{attribute 'qualified_only'}
VAR_GLOBAL
	// PLC Rack
	// Digital Outputs
	bTest					 AT %Q* : BOOL;
	
	// RIO Rack
	// Digital Outputs
	bGreenLight 			AT %Q* : BOOL;
	bRedLight 				AT %Q* : BOOL;
	// Analog Outputs
	nValveOutput 			AT %Q* : INT;
END_VAR

(* stored: Version 1.1.0.1, ProductVersion 3.1.4024.10
   GVL Outputs: Id {8632dc2c-f2e8-400e-b1a8-ffb8dbbb7ffb} *)
